Yaskawa INFORM job: HOME_GUN.JBI

/JOB
//NAME HOME_GUN
///FOLDERNAME HOME
//POS
///NPOS 0,0,0,0,0,1
///TOOL 0
///POSTYPE PULSE
///PULSE
EX00010=56001
//INST
///DATE 2022/06/12 10:02
///ATTR SC,RW
///GROUP1 ST1
NOP
EDTLCK MOVJ EX010 VJ=100.00
END
